# EPICS autosave request: voxtelApp/Db/voxtel_bias_settings.req
$(P)$(R)Voxtel_VP01
$(P)$(R)Voxtel_VP02
$(P)$(R)Voxtel_VP03
$(P)$(R)Voxtel_VP04
$(P)$(R)Voxtel_VP05
$(P)$(R)Voxtel_VP06
$(P)$(R)Voxtel_CC01
$(P)$(R)Voxtel_CC02
$(P)$(R)Voxtel_CC03
$(P)$(R)Voxtel_CC04
$(P)$(R)Voxtel_CC05
$(P)$(R)Voxtel_CC06
$(P)$(R)Voxtel_CC07
$(P)$(R)Voxtel_CC08
$(P)$(R)Voxtel_CC09
$(P)$(R)Voxtel_CC10
$(P)$(R)Voxtel_CC11
$(P)$(R)Voxtel_CC12
$(P)$(R)Voxtel_IREF
$(P)$(R)Voxtel_VV01
$(P)$(R)Voxtel_VV02
$(P)$(R)Voxtel_VV03
$(P)$(R)Voxtel_VV04
$(P)$(R)Voxtel_VV05
$(P)$(R)Voxtel_VV06
$(P)$(R)Voxtel_VV07
$(P)$(R)Voxtel_VV08
$(P)$(R)Voxtel_VV09
$(P)$(R)Voxtel_VV10
